FUNCTION_BLOCK UNIT_Facade (* OPC UA object of the unit (composite skill): PackML unit commands, occupation commands, published unit/occupation state. Replaces the former FC_ControlPort *)
  (* Standard: 61499-2 *)
  (* Version 2.0, 2026-09-27, Project contributors, Filling cell reference model *)
  PACKAGE fillingcell;
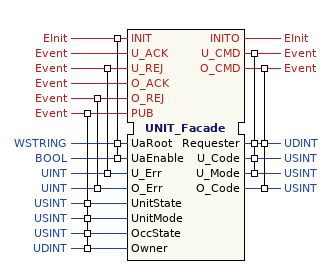
  EVENT_INPUT
    INIT : EInit WITH UaRoot, UaEnable;
    U_ACK;
    U_REJ WITH U_Err;
    O_ACK;
    O_REJ WITH O_Err;
    PUB WITH UnitState, UnitMode, OccState, Owner;
  END_EVENT
  EVENT_OUTPUT
    INITO : EInit;
    U_CMD WITH Requester, U_Code, U_Mode;
    O_CMD WITH Requester, O_Code;
  END_EVENT
  VAR_INPUT
    UaRoot : WSTRING;
    UaEnable : BOOL;
    U_Err : UINT := 4;
    O_Err : UINT := 5;
    UnitState : USINT;
    UnitMode : USINT;
    OccState : USINT;
    Owner : UDINT;
  END_VAR
  VAR_OUTPUT
    Requester : UDINT;
    U_Code : USINT;
    U_Mode : USINT;
    O_Code : USINT;
  END_VAR
  FBS
    Ids : fillingcell::UA_UnitIds;
    Calls : fillingcell::UA_UnitMux;
    Srv_Reset : iec61499::net::SERVER_2_2;
    Srv_Start : iec61499::net::SERVER_2_1;
    Srv_Hold : iec61499::net::SERVER_2_1;
    Srv_Unhold : iec61499::net::SERVER_2_1;
    Srv_Stop : iec61499::net::SERVER_2_1;
    Srv_Abort : iec61499::net::SERVER_2_1;
    Srv_Clear : iec61499::net::SERVER_2_1;
    Srv_Suspend : iec61499::net::SERVER_2_1;
    Srv_Unsuspend : iec61499::net::SERVER_2_1;
    Srv_Occupy : iec61499::net::SERVER_2_1;
    Srv_Release : iec61499::net::SERVER_2_1;
    Srv_Local : iec61499::net::SERVER_2_1;
    Srv_Prioritize : iec61499::net::SERVER_2_1;
    Srv_Remote : iec61499::net::SERVER_2_1;
    Publisher : iec61499::net::PUBLISH_4;
  END_FBS
  EVENT_CONNECTIONS
    Srv_Reset.IND TO Calls.IND_Reset;
    Calls.RSP_Reset TO Srv_Reset.RSP;
    Srv_Start.IND TO Calls.IND_Start;
    Calls.RSP_Start TO Srv_Start.RSP;
    Srv_Hold.IND TO Calls.IND_Hold;
    Calls.RSP_Hold TO Srv_Hold.RSP;
    Srv_Unhold.IND TO Calls.IND_Unhold;
    Calls.RSP_Unhold TO Srv_Unhold.RSP;
    Srv_Stop.IND TO Calls.IND_Stop;
    Calls.RSP_Stop TO Srv_Stop.RSP;
    Srv_Abort.IND TO Calls.IND_Abort;
    Calls.RSP_Abort TO Srv_Abort.RSP;
    Srv_Clear.IND TO Calls.IND_Clear;
    Calls.RSP_Clear TO Srv_Clear.RSP;
    Srv_Suspend.IND TO Calls.IND_Suspend;
    Calls.RSP_Suspend TO Srv_Suspend.RSP;
    Srv_Unsuspend.IND TO Calls.IND_Unsuspend;
    Calls.RSP_Unsuspend TO Srv_Unsuspend.RSP;
    Srv_Occupy.IND TO Calls.IND_Occupy;
    Calls.RSP_Occupy TO Srv_Occupy.RSP;
    Srv_Release.IND TO Calls.IND_Release;
    Calls.RSP_Release TO Srv_Release.RSP;
    Srv_Local.IND TO Calls.IND_Local;
    Calls.RSP_Local TO Srv_Local.RSP;
    Srv_Prioritize.IND TO Calls.IND_Prioritize;
    Calls.RSP_Prioritize TO Srv_Prioritize.RSP;
    Srv_Remote.IND TO Calls.IND_Remote;
    Calls.RSP_Remote TO Srv_Remote.RSP;
    INIT TO Ids.INIT;
    Ids.INITO TO Srv_Reset.INIT;
    Srv_Reset.INITO TO Srv_Start.INIT;
    Srv_Start.INITO TO Srv_Hold.INIT;
    Srv_Hold.INITO TO Srv_Unhold.INIT;
    Srv_Unhold.INITO TO Srv_Stop.INIT;
    Srv_Stop.INITO TO Srv_Abort.INIT;
    Srv_Abort.INITO TO Srv_Clear.INIT;
    Srv_Clear.INITO TO Srv_Suspend.INIT;
    Srv_Suspend.INITO TO Srv_Unsuspend.INIT;
    Srv_Unsuspend.INITO TO Srv_Occupy.INIT;
    Srv_Occupy.INITO TO Srv_Release.INIT;
    Srv_Release.INITO TO Srv_Local.INIT;
    Srv_Local.INITO TO Srv_Prioritize.INIT;
    Srv_Prioritize.INITO TO Srv_Remote.INIT;
    Srv_Remote.INITO TO Publisher.INIT;
    Publisher.INITO TO INITO;
    PUB TO Publisher.REQ;
    Calls.U_CMD TO U_CMD;
    U_ACK TO Calls.U_ACK;
    U_REJ TO Calls.U_REJ;
    Calls.O_CMD TO O_CMD;
    O_ACK TO Calls.O_ACK;
    O_REJ TO Calls.O_REJ;
  END_CONNECTIONS
  DATA_CONNECTIONS
    UaEnable TO Srv_Reset.QI;
    Ids.Id_Reset TO Srv_Reset.ID;
    Srv_Reset.RD_1 TO Calls.Req_Reset;
    Srv_Reset.RD_2 TO Calls.Reset_Mode;
    Calls.Accepted TO Srv_Reset.SD_1;
    Calls.ErrorID TO Srv_Reset.SD_2;
    UaEnable TO Srv_Start.QI;
    Ids.Id_Start TO Srv_Start.ID;
    Srv_Start.RD_1 TO Calls.Req_Start;
    Calls.Accepted TO Srv_Start.SD_1;
    Calls.ErrorID TO Srv_Start.SD_2;
    UaEnable TO Srv_Hold.QI;
    Ids.Id_Hold TO Srv_Hold.ID;
    Srv_Hold.RD_1 TO Calls.Req_Hold;
    Calls.Accepted TO Srv_Hold.SD_1;
    Calls.ErrorID TO Srv_Hold.SD_2;
    UaEnable TO Srv_Unhold.QI;
    Ids.Id_Unhold TO Srv_Unhold.ID;
    Srv_Unhold.RD_1 TO Calls.Req_Unhold;
    Calls.Accepted TO Srv_Unhold.SD_1;
    Calls.ErrorID TO Srv_Unhold.SD_2;
    UaEnable TO Srv_Stop.QI;
    Ids.Id_Stop TO Srv_Stop.ID;
    Srv_Stop.RD_1 TO Calls.Req_Stop;
    Calls.Accepted TO Srv_Stop.SD_1;
    Calls.ErrorID TO Srv_Stop.SD_2;
    UaEnable TO Srv_Abort.QI;
    Ids.Id_Abort TO Srv_Abort.ID;
    Srv_Abort.RD_1 TO Calls.Req_Abort;
    Calls.Accepted TO Srv_Abort.SD_1;
    Calls.ErrorID TO Srv_Abort.SD_2;
    UaEnable TO Srv_Clear.QI;
    Ids.Id_Clear TO Srv_Clear.ID;
    Srv_Clear.RD_1 TO Calls.Req_Clear;
    Calls.Accepted TO Srv_Clear.SD_1;
    Calls.ErrorID TO Srv_Clear.SD_2;
    UaEnable TO Srv_Suspend.QI;
    Ids.Id_Suspend TO Srv_Suspend.ID;
    Srv_Suspend.RD_1 TO Calls.Req_Suspend;
    Calls.Accepted TO Srv_Suspend.SD_1;
    Calls.ErrorID TO Srv_Suspend.SD_2;
    UaEnable TO Srv_Unsuspend.QI;
    Ids.Id_Unsuspend TO Srv_Unsuspend.ID;
    Srv_Unsuspend.RD_1 TO Calls.Req_Unsuspend;
    Calls.Accepted TO Srv_Unsuspend.SD_1;
    Calls.ErrorID TO Srv_Unsuspend.SD_2;
    UaEnable TO Srv_Occupy.QI;
    Ids.Id_Occupy TO Srv_Occupy.ID;
    Srv_Occupy.RD_1 TO Calls.Req_Occupy;
    Calls.Accepted TO Srv_Occupy.SD_1;
    Calls.ErrorID TO Srv_Occupy.SD_2;
    UaEnable TO Srv_Release.QI;
    Ids.Id_Release TO Srv_Release.ID;
    Srv_Release.RD_1 TO Calls.Req_Release;
    Calls.Accepted TO Srv_Release.SD_1;
    Calls.ErrorID TO Srv_Release.SD_2;
    UaEnable TO Srv_Local.QI;
    Ids.Id_Local TO Srv_Local.ID;
    Srv_Local.RD_1 TO Calls.Req_Local;
    Calls.Accepted TO Srv_Local.SD_1;
    Calls.ErrorID TO Srv_Local.SD_2;
    UaEnable TO Srv_Prioritize.QI;
    Ids.Id_Prioritize TO Srv_Prioritize.ID;
    Srv_Prioritize.RD_1 TO Calls.Req_Prioritize;
    Calls.Accepted TO Srv_Prioritize.SD_1;
    Calls.ErrorID TO Srv_Prioritize.SD_2;
    UaEnable TO Srv_Remote.QI;
    Ids.Id_Remote TO Srv_Remote.ID;
    Srv_Remote.RD_1 TO Calls.Req_Remote;
    Calls.Accepted TO Srv_Remote.SD_1;
    Calls.ErrorID TO Srv_Remote.SD_2;
    UaRoot TO Ids.UaRoot;
    UaEnable TO Publisher.QI;
    Ids.IdPub TO Publisher.ID;
    UnitState TO Publisher.SD_1;
    UnitMode TO Publisher.SD_2;
    OccState TO Publisher.SD_3;
    Owner TO Publisher.SD_4;
    U_Err TO Calls.U_Err;
    Calls.U_Code TO U_Code;
    O_Err TO Calls.O_Err;
    Calls.O_Code TO O_Code;
    Calls.U_Mode TO U_Mode;
    Calls.Requester TO Requester;
  END_CONNECTIONS
END_FUNCTION_BLOCK
